// TIA Portal project "Afagyi_nyalna_felmagat" (V15.1)

(* hardware
DEVICE "S7300/ET200M station_1"  S7-300 station
   slot 0: "Rail_0"  Rail  6ES7 390-1***0-0AA0
   slot 2: "PLC_1"  CPU 314C-2 PN/DP  6ES7 314-6EH04-0AB0  V3.3
      slot 2: "PROFINET interface_1"  PN-IO
         slot 1: "Port_1"  Port
         slot 2: "Port_2"  Port
      slot 5: "DI 24/DO 16_1"  DI24/DO16
      slot 6: "AI 5/AO 2_1"  AI5/AO2
      slot 7: "Count_1"  Counter
      slot 8: "Positioning_1"  Positioning
DEVICE "HMI_1"  KTP600 Basic color PN
   slot 0: "HMI_1"  KTP600 Basic color PN  6AV6 647-0AD11-3AX0  12.0.0.0
   slot 1: "HMI_RT_1"  KTP600 Basic color PN  6AV6 647-0AD11-3AX0  12.0.0.0
   slot 5: "HMI_1.IE_CP_1"  PROFINET Interface  12.0.0.0
      slot 1: "PROFINET Interface_1"  PROFINET Interface
         slot 1: "Port_1"  Port
*)

// ===== PLC "PLC_1"  CPU 314C-2 PN/DP =====

DATA_BLOCK "Recept_Lista"   // DB1
{ S7_Optimized_Access := 'FALSE' }
VERSION : 0.1
   VAR
      RECEPT : Array[0..9] of Struct
         Nev : Int;
         Tej : Int;
         Viz : Int;
         Szin : Int;
         Cukor : Int;
      END_STRUCT;
   END_VAR
BEGIN
   RECEPT[0].Nev := 69;
   RECEPT[0].Tej := 69;
   RECEPT[0].Viz := 69;
   RECEPT[0].Szin := 69;
   RECEPT[0].Cukor := 69;
   RECEPT[1].Nev := 69;
   RECEPT[1].Tej := 69;
   RECEPT[1].Viz := 69;
   RECEPT[1].Szin := 69;
   RECEPT[1].Cukor := 69;
   RECEPT[2].Nev := 70;
   RECEPT[2].Tej := 69;
   RECEPT[2].Viz := 100;
   RECEPT[2].Szin := 69;
   RECEPT[2].Cukor := 15;
   RECEPT[3].Nev := 44;
   RECEPT[3].Tej := 16;
   RECEPT[3].Viz := 69;
   RECEPT[3].Szin := 76;
   RECEPT[3].Cukor := 69;
   RECEPT[4].Nev := 432;
   RECEPT[4].Tej := 69;
   RECEPT[4].Viz := 4;
   RECEPT[4].Szin := 69;
   RECEPT[4].Cukor := 345;
   RECEPT[5].Nev := 69;
   RECEPT[5].Tej := 33;
   RECEPT[5].Viz := 69;
   RECEPT[5].Szin := 654;
   RECEPT[5].Cukor := 23;
   RECEPT[6].Nev := 234;
   RECEPT[6].Tej := 69;
   RECEPT[6].Viz := 654;
   RECEPT[6].Szin := 69;
   RECEPT[6].Cukor := 35;
   RECEPT[7].Nev := 69;
   RECEPT[7].Tej := 423;
   RECEPT[7].Viz := 432;
   RECEPT[7].Szin := 69;
   RECEPT[7].Cukor := 43;
   RECEPT[8].Nev := 243;
   RECEPT[8].Tej := 45;
   RECEPT[8].Viz := 69;
   RECEPT[8].Szin := 10;
   RECEPT[8].Cukor := 69;
   RECEPT[9].Nev := 100;
   RECEPT[9].Tej := 25;
   RECEPT[9].Viz := 69;
   RECEPT[9].Szin := 2435;
   RECEPT[9].Cukor := 1;
END_DATA_BLOCK

DATA_BLOCK "Valtozoim"   // DB2
{ S7_Optimized_Access := 'FALSE' }
VERSION : 0.1
   VAR
      Aktualis_receptszam : Int := 1;
      Aktualis_nev : Int;
      Aktualis_tej : Int;
      Aktualis_viz : Int;
      Aktualis_szin : Int;
      Aktualis_cukor : Int;
      Aktualis_regi : Int := 0;
      Mentes : Bool;
   END_VAR
BEGIN
END_DATA_BLOCK

FUNCTION "Betoltes" : Void   // FC1, STL
{ S7_Optimized_Access := 'FALSE' }
VERSION : 0.1
   VAR_TEMP
      adress : DWord;
      X : Int;
      offset : Word;
   END_VAR
BEGIN

REGION Network 1
         L     "Valtozoim".Aktualis_receptszam;  //betoltes
         T     #X;  // int vagy DWORD tipusu Lokalis valtozo
         L     #X;  //   betoltes
         L     1;  // belarakom az 1-et
         -I;
         T     #X;
         L     10;
         *I;
         T     #offset;
   ///  Nev
         L     #offset;
         OPN   "Recept_Lista";
         L     P#0.0;
         L     #offset;

         SLD   3;
         +D;
         T     #adress;
         L     DBW [ #adress];
         OPN   "Valtozoim";
         T     "Valtozoim".Aktualis_nev;
   ///  Tej
         L     #offset;
         L     16#0002;
         +I;
         T     #offset;
         L     #offset;
         OPN   "Recept_Lista";
         L     P#0.0;
         L     #offset;
         SLD   3;
         +D;
         T     #adress;
         L     DBW [ #adress];
         OPN   "Valtozoim";
         T     "Valtozoim".Aktualis_tej;
   /// Viz
         L     #offset;
         L     16#0002;
         +I;
         T     #offset;
         L     #offset;
         OPN   "Recept_Lista";
         L     P#0.0;
         L     #offset;
         SLD   3;
         +D;
         T     #adress;
         L     DBW [ #adress];
         OPN   "Valtozoim";
         T     "Valtozoim".Aktualis_viz;
   ////Szinezek
         L     #offset;
         L     16#0002;
         +I;
         T     #offset;
         L     #offset;
         OPN   "Recept_Lista";
         L     P#0.0;
         L     #offset;
         SLD   3;
         +D;
         T     #adress;
         L     DBW [ #adress];
         OPN   "Valtozoim";
         T     "Valtozoim".Aktualis_szin;
   ////Cukor
         L     #offset;
         L     16#0002;
         +I;
         T     #offset;
         L     #offset;
         OPN   "Recept_Lista";
         L     P#0.0;
         L     #offset;
         SLD   3;
         +D;
         T     #adress;
         L     DBW [ #adress];
         OPN   "Valtozoim";
         T     "Valtozoim".Aktualis_cukor;
END_REGION
END_FUNCTION

FUNCTION "Mentes" : Void   // FC2, STL
{ S7_Optimized_Access := 'FALSE' }
VERSION : 0.1
   VAR_TEMP
      adress : DWord;
      X : Int;
      offset : Word;
   END_VAR
BEGIN

REGION Network 1
   /// nev
         L     "Valtozoim".Aktualis_receptszam;
         T     #X;
         L     #X;
         L     1;
         -I;
         T     #X;
         L     10;
         *I;
         T     #offset;

         L     #offset;
         OPN   "Recept_Lista";
         L     P#0.0;
         L     #offset;

         SLD   3;
         +D;
         T     #adress;
         OPN   "Valtozoim";
         L     "Valtozoim".Aktualis_nev;
         OPN   "Recept_Lista";
         T     DBW [ #adress];

   ////Tej
         L     #offset;
         L     16#0002;
         +I;
         T     #offset;
         L     #offset;
         OPN   "Recept_Lista";
         L     P#0.0;
         L     #offset;
         SLD   3;
         +D;
         T     #adress;
         OPN   "Valtozoim";
         L     "Valtozoim".Aktualis_tej;
         OPN   "Recept_Lista";
         T     DBW [ #adress];

   //// Viz
         L     #offset;
         L     16#0002;
         +I;
         T     #offset;
         L     #offset;
         OPN   "Recept_Lista";
         L     P#0.0;
         L     #offset;
         SLD   3;
         +D;
         T     #adress;
         OPN   "Valtozoim";
         L     "Valtozoim".Aktualis_viz;
         OPN   "Recept_Lista";
         T     DBW [ #adress];

   ////Szinezek
         L     #offset;
         L     16#0002;
         +I;
         T     #offset;
         L     #offset;
         OPN   "Recept_Lista";
         L     P#0.0;
         L     #offset;
         SLD   3;
         +D;
         T     #adress;
         OPN   "Valtozoim";
         L     "Valtozoim".Aktualis_szin;
         OPN   "Recept_Lista";
         T     DBW [ #adress];

   ////Cukor
         L     #offset;
         L     16#0002;
         +I;
         T     #offset;
         L     #offset;
         OPN   "Recept_Lista";
         L     P#0.0;
         L     #offset;
         SLD   3;
         +D;
         T     #adress;
         OPN   "Valtozoim";
         L     "Valtozoim".Aktualis_cukor;
         OPN   "Recept_Lista";
         T     DBW [ #adress];
END_REGION
END_FUNCTION

ORGANIZATION_BLOCK "Main"   // OB1, LAD
TITLE = "Main Program Sweep (Cycle)"
{ S7_Optimized_Access := 'FALSE' }
VERSION : 0.1
   VAR_TEMP
      OB1_EV_CLASS : Byte;   // Bits 0-3 = 1 (Coming event), Bits 4-7 = 1 (Event class 1)
      OB1_SCAN_1 : Byte;   // 1 (Cold restart scan 1 of OB 1), 3 (Scan 2-n of OB 1)
      OB1_PRIORITY : Byte;   // Priority of OB Execution
      OB1_OB_NUMBR : Byte;   // 1 (Organization block 1, OB1)
      OB1_RESERVED_1 : Byte;   // Reserved for system
      OB1_RESERVED_2 : Byte;   // Reserved for system
      OB1_PREV_CYCLE : Int;   // Cycle time of previous OB1 scan (milliseconds)
      OB1_MIN_CYCLE : Int;   // Minimum cycle time of OB1 (milliseconds)
      OB1_MAX_CYCLE : Int;   // Maximum cycle time of OB1 (milliseconds)
      OB1_DATE_TIME : Date_And_Time;   // Date and time OB1 started
   END_VAR
   VAR_TEMP   // added for the SCL form of the ladder/FBD networks
      _w1 : Bool;
   END_VAR
BEGIN

REGION Network 1
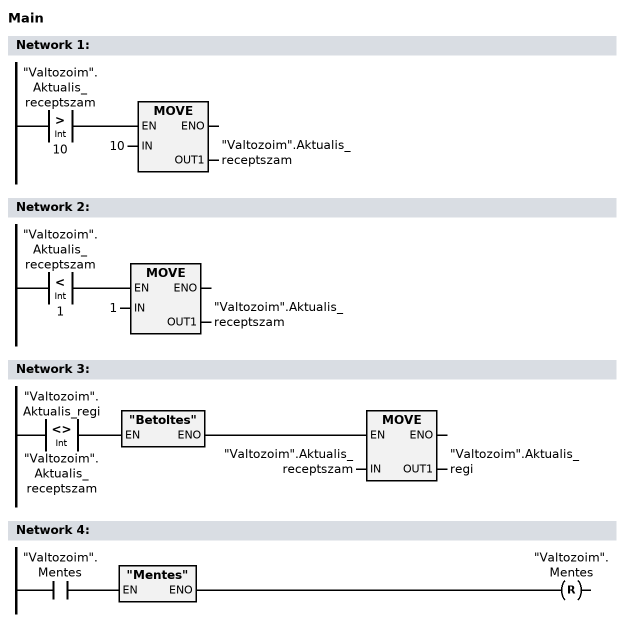
   RUNG wire#powerrail
      { S7_Templates := "SrcType := Int" } GT_Contact(in1 := "Valtozoim".Aktualis_receptszam, in2 := 10)
      { S7_GenerateENO := "TRUE" } Move(in := 10, out1 => "Valtozoim".Aktualis_receptszam)
   END_RUNG
   // the same network as SCL:
   IF "Valtozoim".Aktualis_receptszam > 10 THEN "Valtozoim".Aktualis_receptszam := 10; END_IF;
END_REGION

REGION Network 2
   RUNG wire#powerrail
      { S7_Templates := "SrcType := Int" } LT_Contact(in1 := "Valtozoim".Aktualis_receptszam, in2 := 1)
      { S7_GenerateENO := "TRUE" } Move(in := 1, out1 => "Valtozoim".Aktualis_receptszam)
   END_RUNG
   // the same network as SCL:
   IF "Valtozoim".Aktualis_receptszam < 1 THEN "Valtozoim".Aktualis_receptszam := 1; END_IF;
END_REGION

REGION Network 3
   RUNG wire#powerrail
      { S7_Templates := "SrcType := Int" } NE_Contact(in1 := "Valtozoim".Aktualis_regi, in2 := "Valtozoim".Aktualis_receptszam)
      "Betoltes"()
      { S7_GenerateENO := "TRUE" } Move(in := "Valtozoim".Aktualis_receptszam, out1 => "Valtozoim".Aktualis_regi)
   END_RUNG
   // the same network as SCL:
   "Betoltes"(EN := "Valtozoim".Aktualis_regi <> "Valtozoim".Aktualis_receptszam, ENO => #_w1);
   IF #_w1 THEN "Valtozoim".Aktualis_regi := "Valtozoim".Aktualis_receptszam; END_IF;
END_REGION

REGION Network 4
   RUNG wire#powerrail
      Contact( "Valtozoim".Mentes )
      "Mentes"()
      R_Coil( "Valtozoim".Mentes )
   END_RUNG
   // the same network as SCL:
   "Mentes"(EN := "Valtozoim".Mentes, ENO => #_w1);
   IF #_w1 THEN "Valtozoim".Mentes := FALSE; END_IF;
END_REGION
END_ORGANIZATION_BLOCK

(* ===== HMI "HMI_RT_1" =====
system functions are stored by id; their names below are inferred from use
connection "HMI_Connection_1": ETHERNET, SIMATIC S7 300/400 MPI

HMI tags "Default tag table"
   "Tag_ScreenNumber" : UInt, internal
   "Valtozoim_Aktualis_nev" : Int = PLC Valtozoim.Aktualis_nev AT %DB2.DBW2, 1 s
   "Valtozoim_Aktualis_tej" : Int = PLC Valtozoim.Aktualis_tej AT %DB2.DBW4, 1 s
   "Valtozoim_Aktualis_szin" : Int = PLC Valtozoim.Aktualis_szin AT %DB2.DBW8, 1 s
   "Valtozoim_Aktualis_cukor" : Int = PLC Valtozoim.Aktualis_cukor AT %DB2.DBW10, 1 s
   "Valtozoim_Aktualis_viz" : Int = PLC Valtozoim.Aktualis_viz AT %DB2.DBW6, 1 s
   "Valtozoim_Aktualis_receptszam" : Int = PLC Valtozoim.Aktualis_receptszam AT %DB2.DBW0, 1 s
   "Valtozoim_Mentes" : Bool = PLC Valtozoim.Mentes AT %DB2.DBX14.0, 1 s

Template "Template_1" 320x240
   Button "Exit" at 266,202 size 52x37; TextOff 'Exit'; PictureOff "ExitRuntime_KTP600_Basic_color_PN"; PictureOn "ExitRuntime_KTP600_Basic_color_PN"
      on Release: StopRuntime(0)
   Button "Template_Button" at 213,202 size 52x37; TextOff 'Text'
   Button "Template_Button_1" at 160,202 size 52x37; TextOff 'Text'
   Button "Template_Button_2" at 107,202 size 52x37; TextOff 'Text'
   Button "Start screen" at 54,202 size 52x37; TextOff 'Start screen'; PictureOff "NavigateHome_KTP600_Basic_color_PN"; PictureOn "NavigateHome_KTP600_Basic_color_PN"
      on Release: ActivateScreen("Root screen", 0)
   Button "Alarms" at 1,202 size 52x37; TextOff 'Alarms'; PictureOff "AlarmDisplay_KTP600_Basic_color_PN"; PictureOn "AlarmDisplay_KTP600_Basic_color_PN"
      on Release: function_ef3f5d25("Alarm window_Unacknowledged", -1)
   SymbolicIOField "Symbolic_IO_Field_Screen" at 69,7 size 164x24; TextOff '0'; TextOn '1'; TextList "TextList_ScreenNames"
      ProcessValue <- "Tag_ScreenNumber"
      on Change: ActivateScreenByNumber("Tag_ScreenNumber", 0)
   DateTimeField "HmiScreenItemData" at 235,19 size 85x19
   DateTimeField "HmiScreenItemData_1" at 235,0 size 85x19
   GraphicView "Logo" at 0,0 size 67x38; Picture "Logo of HMI_1"

screen "Root screen" 320x240, template "Template_1"
   on GenerateScreen: SetTag("Tag_ScreenNumber", 1)
   Button "Button_1" at 106,165 size 96x32; TextOff 'Mentés'
      on Click: SetBit("Valtozoim_Mentes")
   IOField "I/O field_3" at 15,159 size 71x25; FormatPattern s99999
      ProcessValue <- "Valtozoim_Aktualis_cukor"
   IOField "I/O field_1" at 115,74 size 71x25; FormatPattern s99999
      ProcessValue <- "Valtozoim_Aktualis_nev"
   IOField "I/O field_2" at 218,159 size 71x25; FormatPattern s99999
      ProcessValue <- "Valtozoim_Aktualis_szin"
   IOField "I/O field_4" at 15,96 size 71x25; FormatPattern s99999
      ProcessValue <- "Valtozoim_Aktualis_viz"
   IOField "I/O field_5" at 218,96 size 71x25; FormatPattern s99999
      ProcessValue <- "Valtozoim_Aktualis_tej"
   IOField "I/O field_6" at 131,129 size 38x25; FormatPattern s99
      ProcessValue <- "Valtozoim_Aktualis_receptszam"
   TextField "Text field_1" at 109,107 size 93x18; Text 'Recept száma'
   TextField "Text field_2" at 131,55 size 26x18; Text 'Név'
   TextField "Text field_3" at 41,69 size 21x18; Text 'Víz'
   TextField "Text field_4" at 237,69 size 21x18; Text 'Tej'
   TextField "Text field_5" at 41,136 size 39x18; Text 'Cukor'
   TextField "Text field_6" at 232,136 size 51x18; Text 'Színező'
   TextField "HmiScreenItemData" at 24,31 size 256x30; Text 'Fagyi Műhely'
*)